INTERFACE ITF_Component_HMI

END_INTERFACE

(* stored: Version 1.1.0.1, ProductVersion 3.1.4024.15
   Itf ITF_Component_HMI: Id {53d14405-dc04-4c14-986c-e6dfca1c6596} *)
